(* CODESYS project CtaAppRefrigants_1.0.0.0.library
   Description: Kältmittel Library der CTA
   Version: 1.0.0.0
   Title: CtaAppRefrigants
   Author: SIS
   LanguageModelAttribute: qualified-access-only
   DocFormat: reStructuredText
   Placeholder: CtaAppRefrigants
   DefaultNamespace: CtaAppRefrigants
   CompiledLibraryCompatibilityVersion: CODESYS V3.5 SP16 Patch 3
   Company: CTA

Project tree, tasks and I/O mapping:
  libraries: CtaSysSensorReCalculation, 1.0.0.0 (CTA); CtaSysConfig, 1.0.0.0 (CTA)
  40 Visualizations/
  00000000-0000-0000-0000-000000000000|D:\CoDeSys\LibrariesV3\trunk\Intern\CAA\CAA Template\3.4.0.0 draft\Placeholder.xml
  00000000-0000-0000-0000-000000000000|D:\CoDeSys\LibrariesV3\trunk\Intern\CAA\CAA Template\3.2.0.3 draft\Prefix.pdf
  00000000-0000-0000-0000-000000000000|D:\CoDeSys\LibrariesV3\trunk\Intern\CAA\CAA Template\3.5.2.0 draft\Placeholder.xml
  20 Structs/
    data type enGas
  50 Images/
  10 Documenation/
    global variables VersionHistory
    global variables readMe
  21 Interface/
  11 Library Parameter/
    global variables Parameter
  12 Konstanten/
  60 Textlisten/
    text list GAS
  13 Globale Variablen/
    global variables GVL_REFRIGANTS
  text list GlobalTextList
  5ce3da45-db07-42e7-a21c-a00fff4ed8f6|C:\Users\sis\Downloads\dip-switch.svg
  5ce3da45-db07-42e7-a21c-a00fff4ed8f6|C:\Users\sis\Downloads\lightning-bolt-circle.svg
  30 Program Organization Units/
    function fcPressToTemp [ST]
    function fcPressToTemp_UserDefined [ST]
    function block FB_BAR_TO_TEMP_SRC [ST]: CALCULATET_VALUE, VALUE, FB_INIT
    function block FB_COURRENT_REFRIGANT [ST]
  5ce3da45-db07-42e7-a21c-a00fff4ed8f6|C:\Users\sis\Downloads\sine-wave.svg
  5ce3da45-db07-42e7-a21c-a00fff4ed8f6|C:\Users\sis\Downloads\eye.svg
  5ce3da45-db07-42e7-a21c-a00fff4ed8f6|C:\Users\sis\Downloads\lan.svg
*)

// 20 Structs/enGas
{attribute 'qualified_only'}
{attribute 'to_string'}
TYPE enGas :
(
R22		       := 0	,
R134a	       := 1	,
R404a	       := 2	,
R407c	       := 3	,
R410a	       := 4	,
R507a          := 5	,
R290	       := 6	,
R600	       := 7	,
R600a	       := 8	,
R717	       := 9	,
R744	       := 10,
R728	       := 11,
R1270	       := 12,
R417A	       := 13,
R422D	       := 14,
R413A	       := 15,
R422A	       := 16,
R423A	       := 17,
R407A	       := 18,
R427A	       := 19,
R245FA         := 20,
R407F	       := 21,
R32            := 22,
HTR01	       := 23,
HTR02	       := 24,
R23            := 25,
HFO1234yf      := 26,
HFO1234ze      := 27,
R455A          := 28,
R170           := 29,
R442A		   := 30,
R447A		   := 31,
R448A		   := 32,
R449A		   := 33,
R450A		   := 34,
R452A		   := 35,
R508B		   := 36,
R452B		   := 37,
R513A		   := 38,
R454B		   := 39);
END_TYPE

// 10 Documenation/VersionHistory
(* 

.. image:: ../../Images/CTA_Logo.jpg
   :align: right
   :width: 15% 

**Vorlage**   


============ =========== =========== ============================================
**Date**     **Version** **Author**  **Change**
------------ ----------- ----------- --------------------------------------------
04.03.2021   0.0.0.0     SIS         Vorlage erstellt

============ =========== =========== ============================================


*)
VAR_GLOBAL
    stInfo : STRING:= '0.0.0.0, Vorlage, CTA';
END_VAR

// 10 Documenation/readMe
(*

**ReadMe**
 
|	**Empfehlung**
|
|	Dokumentrieren Sie die Library für eine nachhaltige Entwicklung
|     
| *Beispiel*
| 
| Dies ist die Vorlage Library der CTA. Erstellen Sie ihre Library anhand dieser Vorlage.
*)

VAR_GLOBAL
    xReadMeDone              :   BOOL;
END_VAR

// 11 Library Parameter/Parameter
{attribute 'qualified_only'}
VAR_GLOBAL CONSTANT
	ATMOSPHERIC_PRESSURE 		: REAL 	:= 1.01325;
END_VAR

// 13 Globale Variablen/GVL_REFRIGANTS
{attribute 'qualified_only'}
VAR_GLOBAL
	FB_COURRENT_REFRIGANT	:	FB_COURRENT_REFRIGANT;
END_VAR

// 30 Program Organization Units/fcPressToTemp
FUNCTION fcPressToTemp : REAL
(* ---------------------------------------------------------------------

	Arguments:
		Gas_Number				Int type
			ID	sigla	name						Mixtured gas: there's the specific bubble temperature table
			------------------------------------------------
			0	R22		    Clorodifluorometano
			1	R134a	    1,1,1,2-tetrafluoroetano
			2	R404a	    							yes
			3	R407c	    							yes
			4	R410a	    							yes
			5	R507a       
			6	R290	    Propano
			7	R600	    Butano
			8	R600a	    2-metil propano (isobutano)
			9	R717	    Ammoniaca
			10	R744	    Anidride carbonica
			11	R728	    Azoto
			12	R1270	    Propilene
			13	R417A	    Isceon MO59					yes
			14	R422D	    Isceon MO29					yes
			15	R413A	    Isceon MO49					yes
			16	R422A	    Isceon MO79					yes
			17	R423A	    Isceon 39TC					yes
			18	R407A	    							yes
			19	R427A	    Forane FX100				yes
			20	R245FA      
			21	R407F	    							yes
			22	R32         
			23	HTR01	    							yes
			24	HTR02	    							yes
			25  R23         
			26  HFO1234yf
			27  HFO1234ze		
			28	R455A
			29	R170
			30	R442A								yes
			31	R447A								yes
			32	R448A								yes
			33	R449A								yes
			34	R450A								yes
			35	R452A								yes
			36	R508B								yes
			37	R452B								yes
			38	R513A								yes
			39	R454B								yes
		
		DewBub					bool type
			DewBub = 0 => DEW temperature
			DewBub = 1 => BUBBLE temperature


	Returns:
		Gas_K_Value[0..5]		real type
			Gas_K_Value[0]
			Gas_K_Value[1]
			Gas_K_Value[2]
			Gas_K_Value[3]
			Gas_K_Value[4]
			Gas_K_Value[5]
	--------------------------------------------------------------------- *)
		
VAR_INPUT
	rBarGas    	: REAL;
	xBubble  	: BOOL;
END_VAR	
	
VAR
	Gas_K_Vect : ARRAY [0..5] OF REAL;
	P_ABS : REAL;
	ka : REAL;
	kb : REAL;
	kc : REAL;
	kd : REAL;
	ke : REAL;
	kf : REAL;
	lnVal : REAL;
	lnVal2 : REAL;
	lnVal3 : REAL;
	lnVal4 : REAL;
	lnVal5 : REAL;
END_VAR

CASE GVL_REFRIGANTS.FB_COURRENT_REFRIGANT.enGasType OF
		0:
		(*
		numero d'ordine :		0
		nome gas :				Clorodifluorometano
		sigla gas :				R22
		T [??C] nell'intervallo:	-50,T(Critica)
		*)
		Gas_K_Vect[0]:= -41.1096482264205;
		Gas_K_Vect[1]:=  21.2819306322367;
		Gas_K_Vect[2]:=   2.44065272718116;
		Gas_K_Vect[3]:=  -0.0249317282670474;
		Gas_K_Vect[4]:=   0.136688844671541;
		Gas_K_Vect[5]:=  -0.0149071222643955;
		
		1:
		(*
		numero d'ordine :		1
		nome gas :				1,1,1,2-tetrafluoroetano
		sigla gas :				R134a
		T [??C] nell'intervallo:	-50,T(Critica)
		*)
		Gas_K_Vect[0]:= -26.3471467442793;
		Gas_K_Vect[1]:=  21.8452905582183;
		Gas_K_Vect[2]:=   2.20366783982819;
		Gas_K_Vect[3]:=   0.199632603006818;
		Gas_K_Vect[4]:=   0.0698503972941902;
		Gas_K_Vect[5]:=  -0.00985258905159315;

		2:
		(*
		numero d'ordine :		2
		nome gas :
		sigla gas :				R404a
		T [??C] nell'intervallo:	-50,T(Critica)
		*)
		IF (xBubble = FALSE) THEN		(* DEW *)
			Gas_K_Vect[0]:= -45.748901093787;
			Gas_K_Vect[1]:=  20.5967151823072;
			Gas_K_Vect[2]:=   2.51284419967593;
			Gas_K_Vect[3]:=  -0.0945527965383469;
			Gas_K_Vect[4]:=   0.162841888195113;
			Gas_K_Vect[5]:=  -0.0207465008241783;
		ELSIF (xBubble = TRUE) THEN		(* BUBBLE *)
			Gas_K_Vect[0]:= -46.4983493820651;
			Gas_K_Vect[1]:=  20.7202160279509;
			Gas_K_Vect[2]:=   2.50734412065389;
			Gas_K_Vect[3]:=  -0.0769875990066375;
			Gas_K_Vect[4]:=   0.152952285317671;
			Gas_K_Vect[5]:=  -0.0189396313974649;	
		END_IF;
		
		3:
		(*
		numero d'ordine :		3
		nome gas :
		sigla gas :				R407c
		T [??C] nell'intervallo:	-50,T(Critica)
		*)
		IF (xBubble = FALSE) THEN		(* DEW *)	
			Gas_K_Vect[0]:= -36.910112428876;
			Gas_K_Vect[1]:=  20.4457088643842;
			Gas_K_Vect[2]:=   2.15351676728359;
			Gas_K_Vect[3]:=   0.0232269981609764;
			Gas_K_Vect[4]:=   0.13033081658634;
			Gas_K_Vect[5]:=  -0.0187558181335497;
		ELSIF (xBubble = TRUE) THEN		(* BUBBLE *)
			Gas_K_Vect[0]:= -43.9022462820594;
			Gas_K_Vect[1]:=  20.7341460204482;
			Gas_K_Vect[2]:=   2.19576841518401;
			Gas_K_Vect[3]:=   0.169790906184501;
			Gas_K_Vect[4]:=   0.0458576682838996;
			Gas_K_Vect[5]:=  -0.00242758479865738;
		END_IF;
		
		4:
		(*
		numero d'ordine :		4
		nome gas :
		sigla gas :				R410a
		T [??C] nell'intervallo:	-50,T(Critica)
		*)
		IF (xBubble = FALSE) THEN		(* DEW *)
			Gas_K_Vect[0]:= -51.5826257807516;
			Gas_K_Vect[1]:=  19.3272015574572;
			Gas_K_Vect[2]:=   2.56423426583869;
			Gas_K_Vect[3]:=  -0.232351050276077;
			Gas_K_Vect[4]:=   0.169505119571792;
			Gas_K_Vect[5]:=  -0.018158416409686;
		ELSIF (xBubble = TRUE) THEN		(* BUBBLE *)		
			Gas_K_Vect[0]:= -51.6537660487418;
			Gas_K_Vect[1]:=  19.2807339405428;
			Gas_K_Vect[2]:=   2.6327930369873;
			Gas_K_Vect[3]:=  -0.279234215225609;
			Gas_K_Vect[4]:=   0.181574477893301;
			Gas_K_Vect[5]:=  -0.0191307050788832;
		END_IF;
		
		5:
		(*
		numero d'ordine :		5
		nome gas :
		sigla gas :				R507a
		T [??C] nell'intervallo:	-50,T(Critica)
		*)
		Gas_K_Vect[0]:= -47.0141477970199;
		Gas_K_Vect[1]:=  20.6129158912814;
		Gas_K_Vect[2]:=   2.53181209499373;
		Gas_K_Vect[3]:=  -0.10045172306225;
		Gas_K_Vect[4]:=   0.161023023927942;
		Gas_K_Vect[5]:=  -0.0201283424739816;

		6:
		(*
		numero d'ordine :		6
		nome gas :				Propano
		sigla gas :				R290
		T [??C] nell'intervallo:	-50,T(Critica)
		*)
		Gas_K_Vect[0]:= -42.4035454543709;
		Gas_K_Vect[1]:=  22.5594387109172;
		Gas_K_Vect[2]:=   2.74963140361839;
		Gas_K_Vect[3]:=  -0.066702684049602;
		Gas_K_Vect[4]:=   0.176660369706708;
		Gas_K_Vect[5]:=  -0.0207714203046422;

		7:
		(*
		numero d'ordine :		7
		nome gas :				Butano
		sigla gas :				R600
		T [??C] nell'intervallo:	-50,T(Critica)
		*)
		Gas_K_Vect[0]:= -0.884445721099827;
		Gas_K_Vect[1]:= 26.2004684462062;
		Gas_K_Vect[2]:=  2.82921680493196;
		Gas_K_Vect[3]:=  0.35068591803767;
		Gas_K_Vect[4]:=  0.037818408074662;
		Gas_K_Vect[5]:= -0.00468164676318171;

		8:
		(*
		numero d'ordine :		8
		nome gas :				2-metil propano (isobutano)
		sigla gas :				R600a
		T [??C] nell'intervallo:	-50,T(Critica)
		*)
		Gas_K_Vect[0]:= -11.9745173151553;
		Gas_K_Vect[1]:=  25.3892006359809;
		Gas_K_Vect[2]:=   2.74435992200506;
		Gas_K_Vect[3]:=   0.343959332662906;
		Gas_K_Vect[4]:=   0.0565626186816232;
		Gas_K_Vect[5]:=  -0.00892047743942617;

		9:
		(*
		numero d'ordine :		9
		nome gas :				Ammoniaca
		sigla gas :				R717
		T [??C] nell'intervallo:	-50,T(Critica)
		*)
		Gas_K_Vect[0]:= -33.6064704499102;
		Gas_K_Vect[1]:=  19.9437204996435;
		Gas_K_Vect[2]:=   1.92121570184513;
		Gas_K_Vect[3]:=   0.0625767945218467;
		Gas_K_Vect[4]:=   0.0694062089568988;
		Gas_K_Vect[5]:=  -0.00537580704892587;

		10:
		(*
		numero d'ordine :		10
		nome gas :				Anidride carbonica			
		sigla gas :				R744
		T [??C] nell'intervallo:	-50,T(Critica)
		*)
		Gas_K_Vect[0]:= -68.822052369851;
		Gas_K_Vect[1]:= -19.2576973567152;
		Gas_K_Vect[2]:=  27.0896577867713;
		Gas_K_Vect[3]:=  -8.95145861831552;
		Gas_K_Vect[4]:=   1.63679465252648;
		Gas_K_Vect[5]:=  -0.113037342883596;
			
		11:
		(*
		numero d'ordine :		11
		nome gas :				Azoto
		sigla gas :				R728
		T [??C] nell'intervallo:	-200, -150
		*)
		Gas_K_Vect[0]:= -195.909117762648;
		Gas_K_Vect[1]:=    8.46523992599931;
		Gas_K_Vect[2]:=    1.0197650602314;
		Gas_K_Vect[3]:=    0.0648037807914613;
		Gas_K_Vect[4]:=    0.0391575844282035;
		Gas_K_Vect[5]:=   -0.00436319461799575;
			
		12:
		(*
		numero d'ordine :		12
		nome gas :				Propilene
		sigla gas :				R1270
		T [??C] nell'intervallo:	-50,T(Critica)
		*)
		Gas_K_Vect[0]:= -47.9679171367073;
		Gas_K_Vect[1]:=  21.6954268760056;
		Gas_K_Vect[2]:=   2.97673135817061;
		Gas_K_Vect[3]:=  -0.256979594564916;
		Gas_K_Vect[4]:=   0.217816389643660;
		Gas_K_Vect[5]:=  -0.0235965058548472;
		
		13:
		(*
		numero d'ordine :		13
		nome gas :				Isceon MO59
		sigla gas :				R417A
		T [??C] nell'intervallo:	-50,T(Critica)
		*)
		IF (xBubble = FALSE) THEN		(* DEW *)		
			Gas_K_Vect[0]:= -34.4102867423192;
			Gas_K_Vect[1]:=  20.9507403822036;
			Gas_K_Vect[2]:=   2.20343980056835;
			Gas_K_Vect[3]:=   0.05968085059208;
			Gas_K_Vect[4]:=   0.138248792494884;
			Gas_K_Vect[5]:=  -0.0209008062185918;
		ELSIF (xBubble = TRUE) THEN		(* BUBBLE *)
			Gas_K_Vect[0]:= -39.411752214372;
			Gas_K_Vect[1]:=  21.4623277845921;
			Gas_K_Vect[2]:=   2.31676972125826;
			Gas_K_Vect[3]:=   0.130080045071396;
			Gas_K_Vect[4]:=   0.080198529199265;
			Gas_K_Vect[5]:=  -0.00900870102926557;	
		END_IF;
		
		14:
		(*
		numero d'ordine :		14
		nome gas :				Isceon MO29
		sigla gas :				R422D
		T [??C] nell'intervallo:	-50,T(Critica)
		*)
		IF (xBubble = FALSE) THEN		(* DEW *)			
			Gas_K_Vect[0]:= -38.6265414902658;
			Gas_K_Vect[1]:=  20.5240402889565;
			Gas_K_Vect[2]:=   2.30405221880948;
			Gas_K_Vect[3]:=  -0.0535410705500753;
			Gas_K_Vect[4]:=   0.177743978680423;
			Gas_K_Vect[5]:=  -0.0255834863631109;
		ELSIF (xBubble = TRUE) THEN		(* BUBBLE *)
			Gas_K_Vect[0]:= -43.4738220244582;
			Gas_K_Vect[1]:=  21.1067562183015;
			Gas_K_Vect[2]:=   2.33180464591279;
			Gas_K_Vect[3]:=   0.104273102683311;
			Gas_K_Vect[4]:=   0.0865221333251471;
			Gas_K_Vect[5]:=  -0.00972093201347337;
		END_IF;
		
		15:
		(*
		numero d'ordine :		15
		nome gas :				Isceon MO49
		sigla gas :				R413A
		T [??C] nell'intervallo:	-50,T(Critica)
		*)
		IF (xBubble = FALSE) THEN		(* DEW *)			
			Gas_K_Vect[0]:= -28.1220231758098;
			Gas_K_Vect[1]:=  21.6388166887428;
			Gas_K_Vect[2]:=   2.19575567708678;
			Gas_K_Vect[3]:=   0.184644478870894;
			Gas_K_Vect[4]:=   0.0822709135668781;
			Gas_K_Vect[5]:=  -0.0120393754211404;
		ELSIF (xBubble = TRUE) THEN		(* BUBBLE *)		
			Gas_K_Vect[0]:=  -30.8935011723763;
			Gas_K_Vect[1]:=   22.3724856315836;
			Gas_K_Vect[2]:=   2.23027689457027;
			Gas_K_Vect[3]:=   0.160301327062238;
			Gas_K_Vect[4]:=   0.0843547299884675;
			Gas_K_Vect[5]:=  -0.0116530969849977;
		END_IF;
				
		16:
		(*
		numero d'ordine :		16
		nome gas :				Isceon MO79
		sigla gas :				R422A
		T [??C] nell'intervallo:	-50,T(Critica)
		*)
		IF (xBubble = FALSE) THEN		(* DEW *)
			Gas_K_Vect[0]:= -44.3066828198618;
			Gas_K_Vect[1]:=  20.2280870199993;
			Gas_K_Vect[2]:=   2.50969470952769;
			Gas_K_Vect[3]:=  -0.153267394642142;
			Gas_K_Vect[4]:=   0.194552097252187;
			Gas_K_Vect[5]:=  -0.0257919126077485;	
		ELSIF (xBubble = TRUE) THEN		(* BUBBLE *)
			Gas_K_Vect[0]:= -46.7609778014458;
			Gas_K_Vect[1]:=  20.5974692650384;
			Gas_K_Vect[2]:=   2.48737308505198;
			Gas_K_Vect[3]:=  -0.0672585974521835;
			Gas_K_Vect[4]:=   0.147799174186759;
			Gas_K_Vect[5]:=  -0.0177088089304702;
		END_IF;
				
		17:
		(*
		numero d'ordine :		17
		nome gas :				Isceon 39TC
		sigla gas :				R423A
		T [??C] nell'intervallo:	-50,T(Critica)
		*)
		IF (xBubble = FALSE) THEN		(* DEW *)
			Gas_K_Vect[0]:= -23.7489717641505;
			Gas_K_Vect[1]:=  22.2574988236004;
			Gas_K_Vect[2]:=   2.25642943075029;
			Gas_K_Vect[3]:=   0.23015613666966;
			Gas_K_Vect[4]:=   0.0704619965936229;
			Gas_K_Vect[5]:=  -0.0121765818510345;	
		ELSIF (xBubble = TRUE) THEN		(* BUBBLE *)
			Gas_K_Vect[0]:= -24.4095381220812;
			Gas_K_Vect[1]:=  22.2218005050376;
			Gas_K_Vect[2]:=   2.27554502820651;
			Gas_K_Vect[3]:=   0.23108133126474;
			Gas_K_Vect[4]:=   0.0612459947892625;
			Gas_K_Vect[5]:=  -0.00905611435349778;
		END_IF;
		
		18:
		(*
		numero d'ordine :		18
		nome gas :				
		sigla gas :				R407A
		T [??C] nell'intervallo:	-50,T(Critica)
		*)
		IF (xBubble = FALSE) THEN		(* DEW *)
			Gas_K_Vect[0]:= -38.8776827152069;
			Gas_K_Vect[1]:=  20.2568599061206;
			Gas_K_Vect[2]:=   2.20527371246278;
			Gas_K_Vect[3]:=  -0.0326893176016479;
			Gas_K_Vect[4]:=   0.150183460115149;
			Gas_K_Vect[5]:=  -0.0211198549026933;
		ELSIF (xBubble = TRUE) THEN		(* BUBBLE *)
			Gas_K_Vect[0]:= -45.2799024334657;
			Gas_K_Vect[1]:=  20.5488354779781;
			Gas_K_Vect[2]:=   2.1988837844;
			Gas_K_Vect[3]:=   0.156651005321399;
			Gas_K_Vect[4]:=   0.0508968249250205;
			Gas_K_Vect[5]:=  -0.00323636758619504;
		END_IF;
		
		19:
		(*
		numero d'ordine :		19
		nome gas :				Forane FX100
		sigla gas :				R427A
		T [??C] nell'intervallo:	-50,T(Critica)
		*)
		IF (xBubble = FALSE) THEN		(* DEW *)
			Gas_K_Vect[0]:= -36.4859120011718;
			Gas_K_Vect[1]:=  20.5914267813576;
			Gas_K_Vect[2]:=   2.18134050505742;
			Gas_K_Vect[3]:=   0.0129688253117425;
			Gas_K_Vect[4]:=   0.14211668910917;
			Gas_K_Vect[5]:=  -0.02081388051727;
		ELSIF (xBubble = TRUE) THEN		(* BUBBLE *)
			Gas_K_Vect[0]:= -43.2389085496711;
			Gas_K_Vect[1]:=  20.9634539711676;
			Gas_K_Vect[2]:=   2.23632977626315;
			Gas_K_Vect[3]:=   0.164109174906234;
			Gas_K_Vect[4]:=   0.0519413635570088;
			Gas_K_Vect[5]:=  -0.00355790211170111;
		END_IF;
		
		20:
		(*
		numero d'ordine :		20
		nome gas :				
		sigla gas :				R245FA
		T [??C] nell'intervallo:	-50,T(Critica)
		*)
		Gas_K_Vect[0]:= 14.54686494;
		Gas_K_Vect[1]:= 24.83337288;
		Gas_K_Vect[2]:=  2.64057146;
		Gas_K_Vect[3]:=  0.2963153984;
		Gas_K_Vect[4]:=  0.02006095713;
		Gas_K_Vect[5]:= -0.0009764156261;
		
		21:
		(*
		numero d'ordine :		21
		nome gas :				
		sigla gas :				R407F
		T [??C] nell'intervallo:	-50,T(Critica)
		*)
		IF (xBubble = FALSE) THEN		(* DEW *)
			Gas_K_Vect[0]:= -39.9518119617676;
			Gas_K_Vect[1]:=  20.1163874886374;
			Gas_K_Vect[2]:=   2.26088427393162;
			Gas_K_Vect[3]:=  -0.115865044368602;
			Gas_K_Vect[4]:=   0.177964099068094;
			Gas_K_Vect[5]:=  -0.024257723502966;
		ELSIF (xBubble = TRUE) THEN		(* BUBBLE *)
			Gas_K_Vect[0]:= -46.3288905505793;
			Gas_K_Vect[1]:=  20.4106027914766;
			Gas_K_Vect[2]:=   2.15434758497607;
			Gas_K_Vect[3]:=   0.170659504127186;
			Gas_K_Vect[4]:=   0.0427791949304127;
			Gas_K_Vect[5]:=  -0.00216818154276298;
		END_IF;
		
		22:
		(*
		numero d'ordine :		22
		nome gas :				
		sigla gas :				R32
		T [??C] nell'intervallo:	-50,T(Critica)
		*)
		Gas_K_Vect[0]:= -51.8767397813099;
		Gas_K_Vect[1]:=  19.3529973508505;
		Gas_K_Vect[2]:=   2.39216523036601 ;
		Gas_K_Vect[3]:=  -0.122399345927881;
		Gas_K_Vect[4]:=   0.126780328948762;
		Gas_K_Vect[5]:=  -0.0126463912359517;
		
		23:
		(*
		numero d'ordine :		23
		nome gas :				
		sigla gas :				HTR01
		T [??C] nell'intervallo:	-50,T(Critica)
		*)
		IF (xBubble = FALSE) THEN		(* DEW *)
			Gas_K_Vect[0]:= -13.9463990152852;
			Gas_K_Vect[1]:=  29.294093323671;
			Gas_K_Vect[2]:=  -5.21929416738665;
			Gas_K_Vect[3]:=   5.15001893745733;
			Gas_K_Vect[4]:=  -1.32511517705558;
			Gas_K_Vect[5]:=   0.134998618838696;
		ELSIF (xBubble = TRUE) THEN		(* BUBBLE *)
			Gas_K_Vect[0]:= -12.7848972089013;
			Gas_K_Vect[1]:=  22.4928892450043;
			Gas_K_Vect[2]:=   4.64329058017742;
			Gas_K_Vect[3]:=  -1.08884761621064;
			Gas_K_Vect[4]:=   0.445024272973559;
			Gas_K_Vect[5]:=  -0.048628854374557;
		END_IF;

		24:
		(*
		numero d'ordine :		24
		nome gas :				
		sigla gas :				HTR02
		T [??C] nell'intervallo:	-50,T(Critica)
		*)
		IF (xBubble = FALSE) THEN		(* DEW *)
			Gas_K_Vect[0]:= -13.7081590529273;
			Gas_K_Vect[1]:=  20.2320552243028;
			Gas_K_Vect[2]:=   4.84119362416973;
			Gas_K_Vect[3]:=  -1.33219525014536;
			Gas_K_Vect[4]:=   0.485339500737623;
			Gas_K_Vect[5]:=  -0.0518810559012798;
		ELSIF (xBubble = TRUE) THEN		(* BUBBLE *)
			Gas_K_Vect[0]:= -14.5410660036204;
			Gas_K_Vect[1]:=  20.5764932110363;
			Gas_K_Vect[2]:=   4.26010624367608;
			Gas_K_Vect[3]:=  -0.950438248171918;
			Gas_K_Vect[4]:=   0.369612628363669;
			Gas_K_Vect[5]:=  -0.0380376000629005;
		END_IF;

		25:
		(*
		numero d'ordine :		25
		nome gas :				
		sigla gas :				R23
		T [??C] nell'intervallo: -100, T(critica)
		*)
		Gas_K_Vect[0]:= -82.23758222;
		Gas_K_Vect[1]:= 17.29330756;
		Gas_K_Vect[2]:= 1.752882693;
		Gas_K_Vect[3]:= 0.1442690406;
		Gas_K_Vect[4]:= 0.05756137185;
		Gas_K_Vect[5]:= -0.007240356749;

		26:
		(*
		numero d'ordine :		26
		nome gas :				HFO1234yf
		sigla gas :				
		T [??C] nell'intervallo:
		*)
		Gas_K_Vect[0]:= -29.78055273;
		Gas_K_Vect[1]:=  22.78382298;
		Gas_K_Vect[2]:=   2.387923224;
		Gas_K_Vect[3]:=   0.1831216582;
		Gas_K_Vect[4]:=   0.0932885491;
		Gas_K_Vect[5]:=  -0.01398246908;

		27:
		(*
		numero d'ordine :		27
		nome gas :				HFO1234ze
		sigla gas :				
		T [??C] nell'intervallo:
		*)
		Gas_K_Vect[0]:= -19.24026003;
		Gas_K_Vect[1]:=  22.91751271;
		Gas_K_Vect[2]:=   2.345141295;
		Gas_K_Vect[3]:=   0.2587325888;
		Gas_K_Vect[4]:=   0.05494216453;
		Gas_K_Vect[5]:=  -0.008415498779;
		
		28:
		(*
		numero d'ordine :		28
		nome gas :				R455A
		sigla gas :				
		T [??C] nell'intervallo:
		*)
		IF (xBubble = FALSE) THEN		(* DEW *)
			Gas_K_Vect[0]:= -39.51663862;
			Gas_K_Vect[1]:=  21.06590853;
			Gas_K_Vect[2]:=   2.666368406;
			Gas_K_Vect[3]:=  -0.57882994;
			Gas_K_Vect[4]:=   0.394419012;
			Gas_K_Vect[5]:=  -0.056274907;
		ELSIF (xBubble = TRUE) THEN		(* BUBBLE *)
			Gas_K_Vect[0]:= -52.57858027;
			Gas_K_Vect[1]:=  22.88565912;
			Gas_K_Vect[2]:=  -0.66733979;
			Gas_K_Vect[3]:=   2.326248721;
			Gas_K_Vect[4]:=  -0.616252112;
			Gas_K_Vect[5]:=   0.073597629;
		END_IF;
		
		29:
		(*
		numero d'ordine :		29
		nome gas :				R170
		sigla gas :				
		T [??C] nell'intervallo:
		*)
		Gas_K_Vect[0]:= -88.70093637;
		Gas_K_Vect[1]:=  17.83266418;
		Gas_K_Vect[2]:=   3.106350849;
		Gas_K_Vect[3]:=  -0.527635572;
		Gas_K_Vect[4]:=   0.256835215;
		Gas_K_Vect[5]:=  -0.025812867;
		
		30:
		(*
		numero d'ordine :		30
		nome gas :				
		sigla gas :				R442A
		T [??C] nell'intervallo:	
		*)
		IF (xBubble = FALSE) THEN		(* DEW *)
			Gas_K_Vect[0]:= -40.17112651;
			Gas_K_Vect[1]:=  20.11890992;
			Gas_K_Vect[2]:=   2.412503977;
			Gas_K_Vect[3]:=  -0.305944263;
			Gas_K_Vect[4]:=   0.256417327;
			Gas_K_Vect[5]:=  -0.034783397;
		ELSIF (xBubble = TRUE) THEN		(* BUBBLE *)
			Gas_K_Vect[0]:= -46.72449144;
			Gas_K_Vect[1]:=  20.41943328;
			Gas_K_Vect[2]:=   2.079669987;
			Gas_K_Vect[3]:=   0.238128647;
			Gas_K_Vect[4]:=   0.019157928;
			Gas_K_Vect[5]:=   0.000760265;
		END_IF;
		
		31:
		(*
		numero d'ordine :		31
		nome gas :				
		sigla gas :				R447A
		T [??C] nell'intervallo:	
		*)
		IF (xBubble = FALSE) THEN		(* DEW *)
			Gas_K_Vect[0]:= -45.27206385;
			Gas_K_Vect[1]:=  19.40380123;
			Gas_K_Vect[2]:=   3.123875645;
			Gas_K_Vect[3]:=  -0.766156771;
			Gas_K_Vect[4]:=   0.365842483;
			Gas_K_Vect[5]:=  -0.042341207;
		ELSIF (xBubble = TRUE) THEN		(* BUBBLE *)
			Gas_K_Vect[0]:= -50.01582453;
			Gas_K_Vect[1]:=  20.48724077;
			Gas_K_Vect[2]:=   1.0725352;
			Gas_K_Vect[3]:=   0.902323353;
			Gas_K_Vect[4]:=  -0.187004779;
			Gas_K_Vect[5]:=   0.02301839;
		END_IF;
		
		32:
		(*
		numero d'ordine :		32
		nome gas :				
		sigla gas :				R448A
		T [??C] nell'intervallo:	
		*)
		IF (xBubble = FALSE) THEN		(* DEW *)
			Gas_K_Vect[0]:= -40.55677057;
			Gas_K_Vect[1]:=  20.41869749;
			Gas_K_Vect[2]:=   2.496862997;
			Gas_K_Vect[3]:=  -0.338592467;
			Gas_K_Vect[4]:=   0.273541423;
			Gas_K_Vect[5]:=  -0.037340136;		
		ELSIF (xBubble = TRUE) THEN		(* BUBBLE *)
			Gas_K_Vect[0]:= -46.40443481;
			Gas_K_Vect[1]:=  20.57271223;
			Gas_K_Vect[2]:=   2.079352892;
			Gas_K_Vect[3]:=   0.277126642;
			Gas_K_Vect[4]:=   0.006334161;
			Gas_K_Vect[5]:=   0.002756286;		
		END_IF;
		
		33:
		(*
		numero d'ordine :		33
		nome gas :				
		sigla gas :				R449A
		T [??C] nell'intervallo:	
		*)
		IF (xBubble = FALSE) THEN		(* DEW *)
			Gas_K_Vect[0]:= -40.31177122;
			Gas_K_Vect[1]:=  20.47685738;
			Gas_K_Vect[2]:=   2.485450465;
			Gas_K_Vect[3]:=  -0.32863564;
			Gas_K_Vect[4]:=   0.273557094;
			Gas_K_Vect[5]:=  -0.037761622;
		ELSIF (xBubble = TRUE) THEN		(* BUBBLE *)
			Gas_K_Vect[0]:= -45.98880287;
			Gas_K_Vect[1]:=  20.67167323;
			Gas_K_Vect[2]:=   1.966024242;
			Gas_K_Vect[3]:=   0.384310469;
			Gas_K_Vect[4]:=  -0.029521834;
			Gas_K_Vect[5]:=   0.006796594;
		END_IF;
		
		34:
		(*
		numero d'ordine :		34
		nome gas :				
		sigla gas :				R450A
		T [??C] nell'intervallo:	
		*)
		IF (xBubble = FALSE) THEN		(* DEW *)
			Gas_K_Vect[0]:= -24.49326038;
			Gas_K_Vect[1]:=  22.23666456;
			Gas_K_Vect[2]:=   2.390544343;
			Gas_K_Vect[3]:=   0.245106746;
			Gas_K_Vect[4]:=   0.014892408;
			Gas_K_Vect[5]:=   3.19E-05;
		ELSIF (xBubble = TRUE) THEN		(* BUBBLE *)
			Gas_K_Vect[0]:= -25.26170079;
			Gas_K_Vect[1]:=  22.21317228;
			Gas_K_Vect[2]:=   2.380575218;
			Gas_K_Vect[3]:=   0.247679685;
			Gas_K_Vect[4]:=   0.017147027;
			Gas_K_Vect[5]:=   0.000325564;
		END_IF;
		
		35:
		(*
		numero d'ordine :		35
		nome gas :				
		sigla gas :				R452A
		T [??C] nell'intervallo:	
		*)
		IF (xBubble = FALSE) THEN		(* DEW *)
			Gas_K_Vect[0]:= -43.44625267;
			Gas_K_Vect[1]:=  20.55414365;
			Gas_K_Vect[2]:=   2.767051606;
			Gas_K_Vect[3]:=  -0.506163915;
			Gas_K_Vect[4]:=   0.33365411;
			Gas_K_Vect[5]:=  -0.045299067;
		ELSIF (xBubble = TRUE) THEN		(* BUBBLE *)
			Gas_K_Vect[0]:= -47.20096036;
			Gas_K_Vect[1]:=  20.55325963;
			Gas_K_Vect[2]:=   2.019648387;
			Gas_K_Vect[3]:=   0.353212053;
			Gas_K_Vect[4]:=  -0.014556284;
			Gas_K_Vect[5]:=   0.004893606;
		END_IF;
		
		36:
		(*
		numero d'ordine :		36
		nome gas :				
		sigla gas :				R508B
		T [??C] nell'intervallo:	
		*)
		IF (xBubble = FALSE) THEN		(* DEW *)
			Gas_K_Vect[0]:= -87.38326636;
			Gas_K_Vect[1]:=  17.02925966;
			Gas_K_Vect[2]:=   1.891129737;
			Gas_K_Vect[3]:=   0.098657554;
			Gas_K_Vect[4]:=   0.087325588;
			Gas_K_Vect[5]:=  -0.012591538;
		ELSIF (xBubble = TRUE) THEN		(* BUBBLE *)
			Gas_K_Vect[0]:= -87.83254411;
			Gas_K_Vect[1]:=  17.3583796;
			Gas_K_Vect[2]:=   1.854714799;
			Gas_K_Vect[3]:=   0.078945325;
			Gas_K_Vect[4]:=   0.091703655;
			Gas_K_Vect[5]:=  -0.012728667;
		END_IF;
		
		37:
		(*
		numero d'ordine :		37
		nome gas :				
		sigla gas :				R452B
		T [??C] nell'intervallo:	
		*)
		IF (xBubble = FALSE) THEN		(* DEW *)
			Gas_K_Vect[0]:= -50.00696642;
			Gas_K_Vect[1]:=  19.41561118;
			Gas_K_Vect[2]:=   3.097970716;
			Gas_K_Vect[3]:=  -0.620537545;
			Gas_K_Vect[4]:=   0.296175305;
			Gas_K_Vect[5]:=  -0.03302368;
		ELSIF (xBubble = TRUE) THEN		(* BUBBLE *)
			Gas_K_Vect[0]:= -50.8960194;
			Gas_K_Vect[1]:=  19.58537708;
			Gas_K_Vect[2]:=   2.497758444;
			Gas_K_Vect[3]:=  -0.158298775;
			Gas_K_Vect[4]:=   0.142379673;
			Gas_K_Vect[5]:=  -0.014097918;
		END_IF;
		
		38:
		(*
		numero d'ordine :		38
		nome gas :				
		sigla gas :				R513A
		T [??C] nell'intervallo:	
		*)
		IF (xBubble = FALSE) THEN		(* DEW *)
			Gas_K_Vect[0]:= -29.75943828;
			Gas_K_Vect[1]:=  22.17062511;
			Gas_K_Vect[2]:=   2.305508119;
			Gas_K_Vect[3]:=   0.17794679;
			Gas_K_Vect[4]:=   0.088255508;
			Gas_K_Vect[5]:=  -0.0129799;
		ELSIF (xBubble = TRUE) THEN		(* BUBBLE *)
			Gas_K_Vect[0]:= -29.86421436;
			Gas_K_Vect[1]:=  22.26259949;
			Gas_K_Vect[2]:=   2.291360574;
			Gas_K_Vect[3]:=   0.176737057;
			Gas_K_Vect[4]:=   0.086396643;
			Gas_K_Vect[5]:=  -0.01246062;
		END_IF;
		
		39:
		(*
		numero d'ordine :		39
		nome gas :				
		sigla gas :				R454B
		T [??C] nell'intervallo:	
		*)
		IF (xBubble = FALSE) THEN		(* DEW *)
			Gas_K_Vect[0]:= -49.70000509;
			Gas_K_Vect[1]:=  19.47117624;
			Gas_K_Vect[2]:=   3.12688722;
			Gas_K_Vect[3]:=  -0.644684859;
			Gas_K_Vect[4]:=   0.305786558;
			Gas_K_Vect[5]:=  -0.034289986;
		ELSIF (xBubble = TRUE) THEN		(* BUBBLE *)
			Gas_K_Vect[0]:= -50.72870823;
			Gas_K_Vect[1]:=  19.64976136;
			Gas_K_Vect[2]:=   2.469592179;
			Gas_K_Vect[3]:=  -0.134096099;
			Gas_K_Vect[4]:=   0.135184895;
			Gas_K_Vect[5]:=  -0.013234352;
		END_IF;
	ELSE
		(* default case : Gas_Number Out of range *)
		Gas_K_Vect[0]:= 0.0;
		Gas_K_Vect[1]:= 0.0;
		Gas_K_Vect[2]:= 0.0;
		Gas_K_Vect[3]:= 0.0;
		Gas_K_Vect[4]:= 0.0;
		Gas_K_Vect[5]:= 0.0;
	END_CASE;
		
	ka := Gas_K_Vect[0];
	kb := Gas_K_Vect[1];
	kc := Gas_K_Vect[2];
	kd := Gas_K_Vect[3];
	ke := Gas_K_Vect[4];
	kf := Gas_K_Vect[5];


	P_ABS := rBarGas + Parameter.ATMOSPHERIC_PRESSURE;

	IF P_ABS > 0.0 THEN
		lnVal  := LN(P_ABS);
		lnVal2 := lnVal*lnVal;
		lnVal3 := lnVal2*lnVal;
		lnVal4 := lnVal3*lnVal;
		lnVal5 := lnVal4*lnVal;

		(* Tsat (P) = a+b*ln P + c*(ln P)^2 + d*(ln P)^3 + e*(ln P)^4 + f*(ln P)^5 *)
		fcPressToTemp := ka + kb * lnVal + kc * lnVal2 + kd * lnVal3 + ke * lnVal4 + kf * lnVal5;
	ELSE
		(* Worst case: twice the minimun temperature admitted for R728 (-200??C) *)
		fcPressToTemp := -400.0;
	END_IF;

END_FUNCTION

// 30 Program Organization Units/FB_COURRENT_REFRIGANT
{attribute 'hide'}
FUNCTION_BLOCK FB_COURRENT_REFRIGANT
VAR_INPUT
END_VAR
VAR_OUTPUT
	enGasType		:	enGas;
END_VAR
VAR
	fbConfigFile	:	CtaSysConfig.fbConfigFile;
	fbenGasType		:	CtaSysConfig.fbINT;
END_VAR

fbConfigFile();
fbenGasType(_usiParaNr := 1, itfConfigFb := fbConfigFile, _MinInit := 0,_MaxInit := 39);
enGasType := fbenGasType.proValue;

END_FUNCTION_BLOCK

// 30 Program Organization Units/fcPressToTemp_UserDefined
FUNCTION fcPressToTemp_UserDefined : REAL
(* ---------------------------------------------------------------------

	Arguments:
		Gas_Number				Int type
			ID	sigla	name						Mixtured gas: there's the specific bubble temperature table
			------------------------------------------------
			0	R22		    Clorodifluorometano
			1	R134a	    1,1,1,2-tetrafluoroetano
			2	R404a	    							yes
			3	R407c	    							yes
			4	R410a	    							yes
			5	R507a       
			6	R290	    Propano
			7	R600	    Butano
			8	R600a	    2-metil propano (isobutano)
			9	R717	    Ammoniaca
			10	R744	    Anidride carbonica
			11	R728	    Azoto
			12	R1270	    Propilene
			13	R417A	    Isceon MO59					yes
			14	R422D	    Isceon MO29					yes
			15	R413A	    Isceon MO49					yes
			16	R422A	    Isceon MO79					yes
			17	R423A	    Isceon 39TC					yes
			18	R407A	    							yes
			19	R427A	    Forane FX100				yes
			20	R245FA      
			21	R407F	    							yes
			22	R32         
			23	HTR01	    							yes
			24	HTR02	    							yes
			25  R23         
			26  HFO1234yf
			27  HFO1234ze
			
			28	R455A
			29	R170
			30	R442A								yes
			31	R447A								yes
			32	R448A								yes
			33	R449A								yes
			34	R450A								yes
			35	R452A								yes
			36	R508B								yes
			37	R452B								yes
			38	R513A								yes
			39	R454B								yes
		
		DewBub					bool type
			DewBub = 0 => DEW temperature
			DewBub = 1 => BUBBLE temperature


	Returns:
		Gas_K_Value[0..5]		real type
			Gas_K_Value[0]
			Gas_K_Value[1]
			Gas_K_Value[2]
			Gas_K_Value[3]
			Gas_K_Value[4]
			Gas_K_Value[5]
	--------------------------------------------------------------------- *)
		
VAR_INPUT
	PGas    	: REAL;
	Gas     	: enGas;
	DewBub  	: BOOL;
END_VAR	
	
VAR
	Gas_K_Vect 	: ARRAY [0..5] OF REAL;
	P_ABS 		: REAL;
	ka 			: REAL;
	kb 			: REAL;
	kc 			: REAL;
	kd 			: REAL;
	ke 			: REAL;
	kf 			: REAL;
	lnVal 		: REAL;
	lnVal2 		: REAL;
	lnVal3 		: REAL;
	lnVal4 		: REAL;
	lnVal5 		: REAL;
END_VAR

CASE Gas OF
		0:
		(*
		numero d'ordine :		1
		nome gas :				Clorodifluorometano
		sigla gas :				R22
		T [??C] nell'intervallo:	-50,T(Critica)
		*)
		Gas_K_Vect[0]:= -41.1096482264205;
		Gas_K_Vect[1]:=  21.2819306322367;
		Gas_K_Vect[2]:=   2.44065272718116;
		Gas_K_Vect[3]:=  -0.0249317282670474;
		Gas_K_Vect[4]:=   0.136688844671541;
		Gas_K_Vect[5]:=  -0.0149071222643955;
		
		1:
		(*
		numero d'ordine :		2
		nome gas :				1,1,1,2-tetrafluoroetano
		sigla gas :				R134a
		T [??C] nell'intervallo:	-50,T(Critica)
		*)
		Gas_K_Vect[0]:= -26.3471467442793;
		Gas_K_Vect[1]:=  21.8452905582183;
		Gas_K_Vect[2]:=   2.20366783982819;
		Gas_K_Vect[3]:=   0.199632603006818;
		Gas_K_Vect[4]:=   0.0698503972941902;
		Gas_K_Vect[5]:=  -0.00985258905159315;

		2:
		(*
		numero d'ordine :		3
		nome gas :
		sigla gas :				R404a
		T [??C] nell'intervallo:	-50,T(Critica)
		*)
		IF (DewBub = FALSE) THEN		(* DEW *)
			Gas_K_Vect[0]:= -45.748901093787;
			Gas_K_Vect[1]:=  20.5967151823072;
			Gas_K_Vect[2]:=   2.51284419967593;
			Gas_K_Vect[3]:=  -0.0945527965383469;
			Gas_K_Vect[4]:=   0.162841888195113;
			Gas_K_Vect[5]:=  -0.0207465008241783;
		ELSIF (DewBub = TRUE) THEN		(* BUBBLE *)
			Gas_K_Vect[0]:= -46.4983493820651;
			Gas_K_Vect[1]:=  20.7202160279509;
			Gas_K_Vect[2]:=   2.50734412065389;
			Gas_K_Vect[3]:=  -0.0769875990066375;
			Gas_K_Vect[4]:=   0.152952285317671;
			Gas_K_Vect[5]:=  -0.0189396313974649;	
		END_IF;
		
		3:
		(*
		numero d'ordine :		4
		nome gas :
		sigla gas :				R407c
		T [??C] nell'intervallo:	-50,T(Critica)
		*)
		IF (DewBub = FALSE) THEN		(* DEW *)	
			Gas_K_Vect[0]:= -36.910112428876;
			Gas_K_Vect[1]:=  20.4457088643842;
			Gas_K_Vect[2]:=   2.15351676728359;
			Gas_K_Vect[3]:=   0.0232269981609764;
			Gas_K_Vect[4]:=   0.13033081658634;
			Gas_K_Vect[5]:=  -0.0187558181335497;
		ELSIF (DewBub = TRUE) THEN		(* BUBBLE *)
			Gas_K_Vect[0]:= -43.9022462820594;
			Gas_K_Vect[1]:=  20.7341460204482;
			Gas_K_Vect[2]:=   2.19576841518401;
			Gas_K_Vect[3]:=   0.169790906184501;
			Gas_K_Vect[4]:=   0.0458576682838996;
			Gas_K_Vect[5]:=  -0.00242758479865738;
		END_IF;
		
		4:
		(*
		numero d'ordine :		5
		nome gas :
		sigla gas :				R410a
		T [??C] nell'intervallo:	-50,T(Critica)
		*)
		IF (DewBub = FALSE) THEN		(* DEW *)
			Gas_K_Vect[0]:= -51.5826257807516;
			Gas_K_Vect[1]:=  19.3272015574572;
			Gas_K_Vect[2]:=   2.56423426583869;
			Gas_K_Vect[3]:=  -0.232351050276077;
			Gas_K_Vect[4]:=   0.169505119571792;
			Gas_K_Vect[5]:=  -0.018158416409686;
		ELSIF (DewBub = TRUE) THEN		(* BUBBLE *)		
			Gas_K_Vect[0]:= -51.6537660487418;
			Gas_K_Vect[1]:=  19.2807339405428;
			Gas_K_Vect[2]:=   2.6327930369873;
			Gas_K_Vect[3]:=  -0.279234215225609;
			Gas_K_Vect[4]:=   0.181574477893301;
			Gas_K_Vect[5]:=  -0.0191307050788832;
		END_IF;
		
		5:
		(*
		numero d'ordine :		6
		nome gas :
		sigla gas :				R507a
		T [??C] nell'intervallo:	-50,T(Critica)
		*)
		Gas_K_Vect[0]:= -47.0141477970199;
		Gas_K_Vect[1]:=  20.6129158912814;
		Gas_K_Vect[2]:=   2.53181209499373;
		Gas_K_Vect[3]:=  -0.10045172306225;
		Gas_K_Vect[4]:=   0.161023023927942;
		Gas_K_Vect[5]:=  -0.0201283424739816;

		6:
		(*
		numero d'ordine :		7
		nome gas :				Propano
		sigla gas :				R290
		T [??C] nell'intervallo:	-50,T(Critica)
		*)
		Gas_K_Vect[0]:= -42.4035454543709;
		Gas_K_Vect[1]:=  22.5594387109172;
		Gas_K_Vect[2]:=   2.74963140361839;
		Gas_K_Vect[3]:=  -0.066702684049602;
		Gas_K_Vect[4]:=   0.176660369706708;
		Gas_K_Vect[5]:=  -0.0207714203046422;

		7:
		(*
		numero d'ordine :		8
		nome gas :				Butano
		sigla gas :				R600
		T [??C] nell'intervallo:	-50,T(Critica)
		*)
		Gas_K_Vect[0]:= -0.884445721099827;
		Gas_K_Vect[1]:= 26.2004684462062;
		Gas_K_Vect[2]:=  2.82921680493196;
		Gas_K_Vect[3]:=  0.35068591803767;
		Gas_K_Vect[4]:=  0.037818408074662;
		Gas_K_Vect[5]:= -0.00468164676318171;

		8:
		(*
		numero d'ordine :		9
		nome gas :				2-metil propano (isobutano)
		sigla gas :				R600a
		T [??C] nell'intervallo:	-50,T(Critica)
		*)
		Gas_K_Vect[0]:= -11.9745173151553;
		Gas_K_Vect[1]:=  25.3892006359809;
		Gas_K_Vect[2]:=   2.74435992200506;
		Gas_K_Vect[3]:=   0.343959332662906;
		Gas_K_Vect[4]:=   0.0565626186816232;
		Gas_K_Vect[5]:=  -0.00892047743942617;

		9:
		(*
		numero d'ordine :		10
		nome gas :				Ammoniaca
		sigla gas :				R717
		T [??C] nell'intervallo:	-50,T(Critica)
		*)
		Gas_K_Vect[0]:= -33.6064704499102;
		Gas_K_Vect[1]:=  19.9437204996435;
		Gas_K_Vect[2]:=   1.92121570184513;
		Gas_K_Vect[3]:=   0.0625767945218467;
		Gas_K_Vect[4]:=   0.0694062089568988;
		Gas_K_Vect[5]:=  -0.00537580704892587;

		10:
		(*
		numero d'ordine :		11
		nome gas :				Anidride carbonica			
		sigla gas :				R744
		T [??C] nell'intervallo:	-50,T(Critica)
		*)
		Gas_K_Vect[0]:= -68.822052369851;
		Gas_K_Vect[1]:= -19.2576973567152;
		Gas_K_Vect[2]:=  27.0896577867713;
		Gas_K_Vect[3]:=  -8.95145861831552;
		Gas_K_Vect[4]:=   1.63679465252648;
		Gas_K_Vect[5]:=  -0.113037342883596;
			
		11:
		(*
		numero d'ordine :		12
		nome gas :				Azoto
		sigla gas :				R728
		T [??C] nell'intervallo:	-200, -150
		*)
		Gas_K_Vect[0]:= -195.909117762648;
		Gas_K_Vect[1]:=    8.46523992599931;
		Gas_K_Vect[2]:=    1.0197650602314;
		Gas_K_Vect[3]:=    0.0648037807914613;
		Gas_K_Vect[4]:=    0.0391575844282035;
		Gas_K_Vect[5]:=   -0.00436319461799575;
			
		12:
		(*
		numero d'ordine :		13
		nome gas :				Propilene
		sigla gas :				R1270
		T [??C] nell'intervallo:	-50,T(Critica)
		*)
		Gas_K_Vect[0]:= -47.9679171367073;
		Gas_K_Vect[1]:=  21.6954268760056;
		Gas_K_Vect[2]:=   2.97673135817061;
		Gas_K_Vect[3]:=  -0.256979594564916;
		Gas_K_Vect[4]:=   0.217816389643660;
		Gas_K_Vect[5]:=  -0.0235965058548472;
		
		13:
		(*
		numero d'ordine :		14
		nome gas :				Isceon MO59
		sigla gas :				R417A
		T [??C] nell'intervallo:	-50,T(Critica)
		*)
		IF (DewBub = FALSE) THEN		(* DEW *)		
			Gas_K_Vect[0]:= -34.4102867423192;
			Gas_K_Vect[1]:=  20.9507403822036;
			Gas_K_Vect[2]:=   2.20343980056835;
			Gas_K_Vect[3]:=   0.05968085059208;
			Gas_K_Vect[4]:=   0.138248792494884;
			Gas_K_Vect[5]:=  -0.0209008062185918;
		ELSIF (DewBub = TRUE) THEN		(* BUBBLE *)
			Gas_K_Vect[0]:= -39.411752214372;
			Gas_K_Vect[1]:=  21.4623277845921;
			Gas_K_Vect[2]:=   2.31676972125826;
			Gas_K_Vect[3]:=   0.130080045071396;
			Gas_K_Vect[4]:=   0.080198529199265;
			Gas_K_Vect[5]:=  -0.00900870102926557;	
		END_IF;
		
		14:
		(*
		numero d'ordine :		15
		nome gas :				Isceon MO29
		sigla gas :				R422D
		T [??C] nell'intervallo:	-50,T(Critica)
		*)
		IF (DewBub = FALSE) THEN		(* DEW *)			
			Gas_K_Vect[0]:= -38.6265414902658;
			Gas_K_Vect[1]:=  20.5240402889565;
			Gas_K_Vect[2]:=   2.30405221880948;
			Gas_K_Vect[3]:=  -0.0535410705500753;
			Gas_K_Vect[4]:=   0.177743978680423;
			Gas_K_Vect[5]:=  -0.0255834863631109;
		ELSIF (DewBub = TRUE) THEN		(* BUBBLE *)
			Gas_K_Vect[0]:= -43.4738220244582;
			Gas_K_Vect[1]:=  21.1067562183015;
			Gas_K_Vect[2]:=   2.33180464591279;
			Gas_K_Vect[3]:=   0.104273102683311;
			Gas_K_Vect[4]:=   0.0865221333251471;
			Gas_K_Vect[5]:=  -0.00972093201347337;
		END_IF;
		
		15:
		(*
		numero d'ordine :		16
		nome gas :				Isceon MO49
		sigla gas :				R413A
		T [??C] nell'intervallo:	-50,T(Critica)
		*)
		IF (DewBub = FALSE) THEN		(* DEW *)			
			Gas_K_Vect[0]:= -28.1220231758098;
			Gas_K_Vect[1]:=  21.6388166887428;
			Gas_K_Vect[2]:=   2.19575567708678;
			Gas_K_Vect[3]:=   0.184644478870894;
			Gas_K_Vect[4]:=   0.0822709135668781;
			Gas_K_Vect[5]:=  -0.0120393754211404;
		ELSIF (DewBub = TRUE) THEN		(* BUBBLE *)		
			Gas_K_Vect[0]:=  -30.8935011723763;
			Gas_K_Vect[1]:=   22.3724856315836;
			Gas_K_Vect[2]:=   2.23027689457027;
			Gas_K_Vect[3]:=   0.160301327062238;
			Gas_K_Vect[4]:=   0.0843547299884675;
			Gas_K_Vect[5]:=  -0.0116530969849977;
		END_IF;
				
		16:
		(*
		numero d'ordine :		17
		nome gas :				Isceon MO79
		sigla gas :				R422A
		T [??C] nell'intervallo:	-50,T(Critica)
		*)
		IF (DewBub = FALSE) THEN		(* DEW *)
			Gas_K_Vect[0]:= -44.3066828198618;
			Gas_K_Vect[1]:=  20.2280870199993;
			Gas_K_Vect[2]:=   2.50969470952769;
			Gas_K_Vect[3]:=  -0.153267394642142;
			Gas_K_Vect[4]:=   0.194552097252187;
			Gas_K_Vect[5]:=  -0.0257919126077485;	
		ELSIF (DewBub = TRUE) THEN		(* BUBBLE *)
			Gas_K_Vect[0]:= -46.7609778014458;
			Gas_K_Vect[1]:=  20.5974692650384;
			Gas_K_Vect[2]:=   2.48737308505198;
			Gas_K_Vect[3]:=  -0.0672585974521835;
			Gas_K_Vect[4]:=   0.147799174186759;
			Gas_K_Vect[5]:=  -0.0177088089304702;
		END_IF;
				
		17:
		(*
		numero d'ordine :		18
		nome gas :				Isceon 39TC
		sigla gas :				R423A
		T [??C] nell'intervallo:	-50,T(Critica)
		*)
		IF (DewBub = FALSE) THEN		(* DEW *)
			Gas_K_Vect[0]:= -23.7489717641505;
			Gas_K_Vect[1]:=  22.2574988236004;
			Gas_K_Vect[2]:=   2.25642943075029;
			Gas_K_Vect[3]:=   0.23015613666966;
			Gas_K_Vect[4]:=   0.0704619965936229;
			Gas_K_Vect[5]:=  -0.0121765818510345;	
		ELSIF (DewBub = TRUE) THEN		(* BUBBLE *)
			Gas_K_Vect[0]:= -24.4095381220812;
			Gas_K_Vect[1]:=  22.2218005050376;
			Gas_K_Vect[2]:=   2.27554502820651;
			Gas_K_Vect[3]:=   0.23108133126474;
			Gas_K_Vect[4]:=   0.0612459947892625;
			Gas_K_Vect[5]:=  -0.00905611435349778;
		END_IF;
		
		18:
		(*
		numero d'ordine :		19
		nome gas :				
		sigla gas :				R407A
		T [??C] nell'intervallo:	-50,T(Critica)
		*)
		IF (DewBub = FALSE) THEN		(* DEW *)
			Gas_K_Vect[0]:= -38.8776827152069;
			Gas_K_Vect[1]:=  20.2568599061206;
			Gas_K_Vect[2]:=   2.20527371246278;
			Gas_K_Vect[3]:=  -0.0326893176016479;
			Gas_K_Vect[4]:=   0.150183460115149;
			Gas_K_Vect[5]:=  -0.0211198549026933;
		ELSIF (DewBub = TRUE) THEN		(* BUBBLE *)
			Gas_K_Vect[0]:= -45.2799024334657;
			Gas_K_Vect[1]:=  20.5488354779781;
			Gas_K_Vect[2]:=   2.1988837844;
			Gas_K_Vect[3]:=   0.156651005321399;
			Gas_K_Vect[4]:=   0.0508968249250205;
			Gas_K_Vect[5]:=  -0.00323636758619504;
		END_IF;
		
		19:
		(*
		numero d'ordine :		20
		nome gas :				Forane FX100
		sigla gas :				R427A
		T [??C] nell'intervallo:	-50,T(Critica)
		*)
		IF (DewBub = FALSE) THEN		(* DEW *)
			Gas_K_Vect[0]:= -36.4859120011718;
			Gas_K_Vect[1]:=  20.5914267813576;
			Gas_K_Vect[2]:=   2.18134050505742;
			Gas_K_Vect[3]:=   0.0129688253117425;
			Gas_K_Vect[4]:=   0.14211668910917;
			Gas_K_Vect[5]:=  -0.02081388051727;
		ELSIF (DewBub = TRUE) THEN		(* BUBBLE *)
			Gas_K_Vect[0]:= -43.2389085496711;
			Gas_K_Vect[1]:=  20.9634539711676;
			Gas_K_Vect[2]:=   2.23632977626315;
			Gas_K_Vect[3]:=   0.164109174906234;
			Gas_K_Vect[4]:=   0.0519413635570088;
			Gas_K_Vect[5]:=  -0.00355790211170111;
		END_IF;
		
		20:
		(*
		numero d'ordine :		21
		nome gas :				
		sigla gas :				R245FA
		T [??C] nell'intervallo:	-50,T(Critica)
		*)
		Gas_K_Vect[0]:= 14.54686494;
		Gas_K_Vect[1]:= 24.83337288;
		Gas_K_Vect[2]:=  2.64057146;
		Gas_K_Vect[3]:=  0.2963153984;
		Gas_K_Vect[4]:=  0.02006095713;
		Gas_K_Vect[5]:= -0.0009764156261;
		
		21:
		(*
		numero d'ordine :		22
		nome gas :				
		sigla gas :				R407F
		T [??C] nell'intervallo:	-50,T(Critica)
		*)
		IF (DewBub = FALSE) THEN		(* DEW *)
			Gas_K_Vect[0]:= -39.9518119617676;
			Gas_K_Vect[1]:=  20.1163874886374;
			Gas_K_Vect[2]:=   2.26088427393162;
			Gas_K_Vect[3]:=  -0.115865044368602;
			Gas_K_Vect[4]:=   0.177964099068094;
			Gas_K_Vect[5]:=  -0.024257723502966;
		ELSIF (DewBub = TRUE) THEN		(* BUBBLE *)
			Gas_K_Vect[0]:= -46.3288905505793;
			Gas_K_Vect[1]:=  20.4106027914766;
			Gas_K_Vect[2]:=   2.15434758497607;
			Gas_K_Vect[3]:=   0.170659504127186;
			Gas_K_Vect[4]:=   0.0427791949304127;
			Gas_K_Vect[5]:=  -0.00216818154276298;
		END_IF;
		
		22:
		(*
		numero d'ordine :		23
		nome gas :				
		sigla gas :				R32
		T [??C] nell'intervallo:	-50,T(Critica)
		*)
		Gas_K_Vect[0]:= -51.8767397813099;
		Gas_K_Vect[1]:=  19.3529973508505;
		Gas_K_Vect[2]:=   2.39216523036601 ;
		Gas_K_Vect[3]:=  -0.122399345927881;
		Gas_K_Vect[4]:=   0.126780328948762;
		Gas_K_Vect[5]:=  -0.0126463912359517;
		
		23:
		(*
		numero d'ordine :		24
		nome gas :				
		sigla gas :				HTR01
		T [??C] nell'intervallo:	-50,T(Critica)
		*)
		IF (DewBub = FALSE) THEN		(* DEW *)
			Gas_K_Vect[0]:= -13.9463990152852;
			Gas_K_Vect[1]:=  29.294093323671;
			Gas_K_Vect[2]:=  -5.21929416738665;
			Gas_K_Vect[3]:=   5.15001893745733;
			Gas_K_Vect[4]:=  -1.32511517705558;
			Gas_K_Vect[5]:=   0.134998618838696;
		ELSIF (DewBub = TRUE) THEN		(* BUBBLE *)
			Gas_K_Vect[0]:= -12.7848972089013;
			Gas_K_Vect[1]:=  22.4928892450043;
			Gas_K_Vect[2]:=   4.64329058017742;
			Gas_K_Vect[3]:=  -1.08884761621064;
			Gas_K_Vect[4]:=   0.445024272973559;
			Gas_K_Vect[5]:=  -0.048628854374557;
		END_IF;

		24:
		(*
		numero d'ordine :		25
		nome gas :				
		sigla gas :				HTR02
		T [??C] nell'intervallo:	-50,T(Critica)
		*)
		IF (DewBub = FALSE) THEN		(* DEW *)
			Gas_K_Vect[0]:= -13.7081590529273;
			Gas_K_Vect[1]:=  20.2320552243028;
			Gas_K_Vect[2]:=   4.84119362416973;
			Gas_K_Vect[3]:=  -1.33219525014536;
			Gas_K_Vect[4]:=   0.485339500737623;
			Gas_K_Vect[5]:=  -0.0518810559012798;
		ELSIF (DewBub = TRUE) THEN		(* BUBBLE *)
			Gas_K_Vect[0]:= -14.5410660036204;
			Gas_K_Vect[1]:=  20.5764932110363;
			Gas_K_Vect[2]:=   4.26010624367608;
			Gas_K_Vect[3]:=  -0.950438248171918;
			Gas_K_Vect[4]:=   0.369612628363669;
			Gas_K_Vect[5]:=  -0.0380376000629005;
		END_IF;

		25:
		(*
		numero d'ordine :		26
		nome gas :				
		sigla gas :				R23
		T [??C] nell'intervallo: -100, T(critica)
		*)
		Gas_K_Vect[0]:= -82.23758222;
		Gas_K_Vect[1]:= 17.29330756;
		Gas_K_Vect[2]:= 1.752882693;
		Gas_K_Vect[3]:= 0.1442690406;
		Gas_K_Vect[4]:= 0.05756137185;
		Gas_K_Vect[5]:= -0.007240356749;

		26:
		(*
		numero d'ordine :		27
		nome gas :				HFO1234yf
		sigla gas :				
		T [??C] nell'intervallo:
		*)
		Gas_K_Vect[0]:= -29.78055273;
		Gas_K_Vect[1]:=  22.78382298;
		Gas_K_Vect[2]:=   2.387923224;
		Gas_K_Vect[3]:=   0.1831216582;
		Gas_K_Vect[4]:=   0.0932885491;
		Gas_K_Vect[5]:=  -0.01398246908;

		27:
		(*
		numero d'ordine :		28
		nome gas :				HFO1234ze
		sigla gas :				
		T [??C] nell'intervallo:
		*)
		Gas_K_Vect[0]:= -19.24026003;
		Gas_K_Vect[1]:=  22.91751271;
		Gas_K_Vect[2]:=   2.345141295;
		Gas_K_Vect[3]:=   0.2587325888;
		Gas_K_Vect[4]:=   0.05494216453;
		Gas_K_Vect[5]:=  -0.008415498779;
		
		28:
		(*
		numero d'ordine :		29
		nome gas :				R455A
		sigla gas :				
		T [??C] nell'intervallo:
		*)
		IF (DewBub = FALSE) THEN		(* DEW *)
			Gas_K_Vect[0]:= -39.51663862;
			Gas_K_Vect[1]:=  21.06590853;
			Gas_K_Vect[2]:=   2.666368406;
			Gas_K_Vect[3]:=  -0.57882994;
			Gas_K_Vect[4]:=   0.394419012;
			Gas_K_Vect[5]:=  -0.056274907;
		ELSIF (DewBub = TRUE) THEN		(* BUBBLE *)
			Gas_K_Vect[0]:= -52.57858027;
			Gas_K_Vect[1]:=  22.88565912;
			Gas_K_Vect[2]:=  -0.66733979;
			Gas_K_Vect[3]:=   2.326248721;
			Gas_K_Vect[4]:=  -0.616252112;
			Gas_K_Vect[5]:=   0.073597629;
		END_IF;
		
		29:
		(*
		numero d'ordine :		30
		nome gas :				R170
		sigla gas :				
		T [??C] nell'intervallo:
		*)
		Gas_K_Vect[0]:= -88.70093637;
		Gas_K_Vect[1]:=  17.83266418;
		Gas_K_Vect[2]:=   3.106350849;
		Gas_K_Vect[3]:=  -0.527635572;
		Gas_K_Vect[4]:=   0.256835215;
		Gas_K_Vect[5]:=  -0.025812867;
		
		30:
		(*
		numero d'ordine :		31
		nome gas :				
		sigla gas :				R442A
		T [??C] nell'intervallo:	
		*)
		IF (DewBub = FALSE) THEN		(* DEW *)
			Gas_K_Vect[0]:= -40.17112651;
			Gas_K_Vect[1]:=  20.11890992;
			Gas_K_Vect[2]:=   2.412503977;
			Gas_K_Vect[3]:=  -0.305944263;
			Gas_K_Vect[4]:=   0.256417327;
			Gas_K_Vect[5]:=  -0.034783397;
		ELSIF (DewBub = TRUE) THEN		(* BUBBLE *)
			Gas_K_Vect[0]:= -46.72449144;
			Gas_K_Vect[1]:=  20.41943328;
			Gas_K_Vect[2]:=   2.079669987;
			Gas_K_Vect[3]:=   0.238128647;
			Gas_K_Vect[4]:=   0.019157928;
			Gas_K_Vect[5]:=   0.000760265;
		END_IF;
		
		31:
		(*
		numero d'ordine :		32
		nome gas :				
		sigla gas :				R447A
		T [??C] nell'intervallo:	
		*)
		IF (DewBub = FALSE) THEN		(* DEW *)
			Gas_K_Vect[0]:= -45.27206385;
			Gas_K_Vect[1]:=  19.40380123;
			Gas_K_Vect[2]:=   3.123875645;
			Gas_K_Vect[3]:=  -0.766156771;
			Gas_K_Vect[4]:=   0.365842483;
			Gas_K_Vect[5]:=  -0.042341207;
		ELSIF (DewBub = TRUE) THEN		(* BUBBLE *)
			Gas_K_Vect[0]:= -50.01582453;
			Gas_K_Vect[1]:=  20.48724077;
			Gas_K_Vect[2]:=   1.0725352;
			Gas_K_Vect[3]:=   0.902323353;
			Gas_K_Vect[4]:=  -0.187004779;
			Gas_K_Vect[5]:=   0.02301839;
		END_IF;
		
		32:
		(*
		numero d'ordine :		33
		nome gas :				
		sigla gas :				R448A
		T [??C] nell'intervallo:	
		*)
		IF (DewBub = FALSE) THEN		(* DEW *)
			Gas_K_Vect[0]:= -40.55677057;
			Gas_K_Vect[1]:=  20.41869749;
			Gas_K_Vect[2]:=   2.496862997;
			Gas_K_Vect[3]:=  -0.338592467;
			Gas_K_Vect[4]:=   0.273541423;
			Gas_K_Vect[5]:=  -0.037340136;		
		ELSIF (DewBub = TRUE) THEN		(* BUBBLE *)
			Gas_K_Vect[0]:= -46.40443481;
			Gas_K_Vect[1]:=  20.57271223;
			Gas_K_Vect[2]:=   2.079352892;
			Gas_K_Vect[3]:=   0.277126642;
			Gas_K_Vect[4]:=   0.006334161;
			Gas_K_Vect[5]:=   0.002756286;		
		END_IF;
		
		33:
		(*
		numero d'ordine :		34
		nome gas :				
		sigla gas :				R449A
		T [??C] nell'intervallo:	
		*)
		IF (DewBub = FALSE) THEN		(* DEW *)
			Gas_K_Vect[0]:= -40.31177122;
			Gas_K_Vect[1]:=  20.47685738;
			Gas_K_Vect[2]:=   2.485450465;
			Gas_K_Vect[3]:=  -0.32863564;
			Gas_K_Vect[4]:=   0.273557094;
			Gas_K_Vect[5]:=  -0.037761622;
		ELSIF (DewBub = TRUE) THEN		(* BUBBLE *)
			Gas_K_Vect[0]:= -45.98880287;
			Gas_K_Vect[1]:=  20.67167323;
			Gas_K_Vect[2]:=   1.966024242;
			Gas_K_Vect[3]:=   0.384310469;
			Gas_K_Vect[4]:=  -0.029521834;
			Gas_K_Vect[5]:=   0.006796594;
		END_IF;
		
		34:
		(*
		numero d'ordine :		35
		nome gas :				
		sigla gas :				R450A
		T [??C] nell'intervallo:	
		*)
		IF (DewBub = FALSE) THEN		(* DEW *)
			Gas_K_Vect[0]:= -24.49326038;
			Gas_K_Vect[1]:=  22.23666456;
			Gas_K_Vect[2]:=   2.390544343;
			Gas_K_Vect[3]:=   0.245106746;
			Gas_K_Vect[4]:=   0.014892408;
			Gas_K_Vect[5]:=   3.19E-05;
		ELSIF (DewBub = TRUE) THEN		(* BUBBLE *)
			Gas_K_Vect[0]:= -25.26170079;
			Gas_K_Vect[1]:=  22.21317228;
			Gas_K_Vect[2]:=   2.380575218;
			Gas_K_Vect[3]:=   0.247679685;
			Gas_K_Vect[4]:=   0.017147027;
			Gas_K_Vect[5]:=   0.000325564;
		END_IF;
		
		35:
		(*
		numero d'ordine :		36
		nome gas :				
		sigla gas :				R452A
		T [??C] nell'intervallo:	
		*)
		IF (DewBub = FALSE) THEN		(* DEW *)
			Gas_K_Vect[0]:= -43.44625267;
			Gas_K_Vect[1]:=  20.55414365;
			Gas_K_Vect[2]:=   2.767051606;
			Gas_K_Vect[3]:=  -0.506163915;
			Gas_K_Vect[4]:=   0.33365411;
			Gas_K_Vect[5]:=  -0.045299067;
		ELSIF (DewBub = TRUE) THEN		(* BUBBLE *)
			Gas_K_Vect[0]:= -47.20096036;
			Gas_K_Vect[1]:=  20.55325963;
			Gas_K_Vect[2]:=   2.019648387;
			Gas_K_Vect[3]:=   0.353212053;
			Gas_K_Vect[4]:=  -0.014556284;
			Gas_K_Vect[5]:=   0.004893606;
		END_IF;
		
		36:
		(*
		numero d'ordine :		37
		nome gas :				
		sigla gas :				R508B
		T [??C] nell'intervallo:	
		*)
		IF (DewBub = FALSE) THEN		(* DEW *)
			Gas_K_Vect[0]:= -87.38326636;
			Gas_K_Vect[1]:=  17.02925966;
			Gas_K_Vect[2]:=   1.891129737;
			Gas_K_Vect[3]:=   0.098657554;
			Gas_K_Vect[4]:=   0.087325588;
			Gas_K_Vect[5]:=  -0.012591538;
		ELSIF (DewBub = TRUE) THEN		(* BUBBLE *)
			Gas_K_Vect[0]:= -87.83254411;
			Gas_K_Vect[1]:=  17.3583796;
			Gas_K_Vect[2]:=   1.854714799;
			Gas_K_Vect[3]:=   0.078945325;
			Gas_K_Vect[4]:=   0.091703655;
			Gas_K_Vect[5]:=  -0.012728667;
		END_IF;
		
		37:
		(*
		numero d'ordine :		38
		nome gas :				
		sigla gas :				R452B
		T [??C] nell'intervallo:	
		*)
		IF (DewBub = FALSE) THEN		(* DEW *)
			Gas_K_Vect[0]:= -50.00696642;
			Gas_K_Vect[1]:=  19.41561118;
			Gas_K_Vect[2]:=   3.097970716;
			Gas_K_Vect[3]:=  -0.620537545;
			Gas_K_Vect[4]:=   0.296175305;
			Gas_K_Vect[5]:=  -0.03302368;
		ELSIF (DewBub = TRUE) THEN		(* BUBBLE *)
			Gas_K_Vect[0]:= -50.8960194;
			Gas_K_Vect[1]:=  19.58537708;
			Gas_K_Vect[2]:=   2.497758444;
			Gas_K_Vect[3]:=  -0.158298775;
			Gas_K_Vect[4]:=   0.142379673;
			Gas_K_Vect[5]:=  -0.014097918;
		END_IF;
		
		38:
		(*
		numero d'ordine :		39
		nome gas :				
		sigla gas :				R513A
		T [??C] nell'intervallo:	
		*)
		IF (DewBub = FALSE) THEN		(* DEW *)
			Gas_K_Vect[0]:= -29.75943828;
			Gas_K_Vect[1]:=  22.17062511;
			Gas_K_Vect[2]:=   2.305508119;
			Gas_K_Vect[3]:=   0.17794679;
			Gas_K_Vect[4]:=   0.088255508;
			Gas_K_Vect[5]:=  -0.0129799;
		ELSIF (DewBub = TRUE) THEN		(* BUBBLE *)
			Gas_K_Vect[0]:= -29.86421436;
			Gas_K_Vect[1]:=  22.26259949;
			Gas_K_Vect[2]:=   2.291360574;
			Gas_K_Vect[3]:=   0.176737057;
			Gas_K_Vect[4]:=   0.086396643;
			Gas_K_Vect[5]:=  -0.01246062;
		END_IF;
		
		39:
		(*
		numero d'ordine :		40
		nome gas :				
		sigla gas :				R454B
		T [??C] nell'intervallo:	
		*)
		IF (DewBub = FALSE) THEN		(* DEW *)
			Gas_K_Vect[0]:= -49.70000509;
			Gas_K_Vect[1]:=  19.47117624;
			Gas_K_Vect[2]:=   3.12688722;
			Gas_K_Vect[3]:=  -0.644684859;
			Gas_K_Vect[4]:=   0.305786558;
			Gas_K_Vect[5]:=  -0.034289986;
		ELSIF (DewBub = TRUE) THEN		(* BUBBLE *)
			Gas_K_Vect[0]:= -50.72870823;
			Gas_K_Vect[1]:=  19.64976136;
			Gas_K_Vect[2]:=   2.469592179;
			Gas_K_Vect[3]:=  -0.134096099;
			Gas_K_Vect[4]:=   0.135184895;
			Gas_K_Vect[5]:=  -0.013234352;
		END_IF;
	ELSE
		(* default case : Gas_Number Out of range *)
		Gas_K_Vect[0]:= 0.0;
		Gas_K_Vect[1]:= 0.0;
		Gas_K_Vect[2]:= 0.0;
		Gas_K_Vect[3]:= 0.0;
		Gas_K_Vect[4]:= 0.0;
		Gas_K_Vect[5]:= 0.0;
	END_CASE;
		
	ka := Gas_K_Vect[0];
	kb := Gas_K_Vect[1];
	kc := Gas_K_Vect[2];
	kd := Gas_K_Vect[3];
	ke := Gas_K_Vect[4];
	kf := Gas_K_Vect[5];


	P_ABS := PGas + Parameter.ATMOSPHERIC_PRESSURE;

	IF P_ABS > 0.0 THEN
		lnVal  := LN(P_ABS);
		lnVal2 := lnVal*lnVal;
		lnVal3 := lnVal2*lnVal;
		lnVal4 := lnVal3*lnVal;
		lnVal5 := lnVal4*lnVal;

		(* Tsat (P) = a+b*ln P + c*(ln P)^2 + d*(ln P)^3 + e*(ln P)^4 + f*(ln P)^5 *)
		fcPressToTemp_UserDefined := ka + kb * lnVal + kc * lnVal2 + kd * lnVal3 + ke * lnVal4 + kf * lnVal5;
	ELSE
		(* Worst case: twice the minimun temperature admitted for R728 (-200??C) *)
		fcPressToTemp_UserDefined := -400.0;
	END_IF;

END_FUNCTION

// 30 Program Organization Units/FB_BAR_TO_TEMP_SRC
FUNCTION_BLOCK FB_BAR_TO_TEMP_SRC EXTENDS CtaSysSensorReCalculation.FB_SENSOR_RE_CALCULATE
VAR_INPUT
	xBubble		:	BOOL;
END_VAR

PROPERTY CALCULATET_VALUE : REAL
GET
rCalculatet := fcPressToTemp(rBarGas := rValue,xBubble := xBubble);
CALCULATET_VALUE := rCalculatet;
END_GET
END_PROPERTY

PROPERTY VALUE : REAL
SET
rValue := VALUE;
END_SET
END_PROPERTY

//FB_Init ist immer implizit verfügbar und wird primär für die Initialisierung verwendet.
//Der Rückgabewert wird nicht ausgewertet. Für gezielte Einflussnahme können Sie
//die Methoden explizit deklarieren und darin mit dem Standard-Initialisierungscode 
//zusätzlichen Code bereitstellen. Sie können den Rückgabewert auswerten.
METHOD FB_Init: BOOL
VAR_INPUT    
	bInitRetains: BOOL; // TRUE: Die Retain-Variablen werden initialisiert (Reset warm / Reset kalt)    
	bInCopyCode	: BOOL;  // TRUE: Die Instanz wird danach in den Kopiercode kopiert (Online-Change)
	_stUnit		: STRING(5);
	_xBubble	: BOOL;
END_VAR
xBubble := _xBubble;
stUNIT	:= _stUnit;
END_METHOD

END_FUNCTION_BLOCK

(* text list GAS (id | default)
  R22 | R22
  R134a | R134a
  R404a | R404a
  R407c | R407c
  R410a | R410a
  R507a | R507a
  R290 | R290
  R600 | R600
  R600a | R600a
  R717 | R717
  R744 | R744
  R728 | R728
  R1270 | R1270
  R417A | R417A
  R422D | R422D
  R413A | R413A
  R422A | R422A
  R423A | R423A
  R407A | R407A
  R427A | R427A
  R245FA | R245FA
  R407F | R407F
  R32 | R32
  HTR01 | HTR01
  HTR02 | HTR02
  R23 | R23
  HFO1234yf | HFO1234yf
  HFO1234ze | HFO1234ze
  R455A | R455A
  R170 | R170
  R442A | R442A
  R447A | R447A
  R448A | R448A
  R449A | R449A
  R450A | R450A
  R452A | R452A
  R508B | R508B
  R452B | R452B
  R513A | R513A
  R454B | R454B
   |  *)
